% RSLogix 500 project Pump Control HOA and Alarms.RSS, saved by version 8.30.00.16 %
PROJECT "SIM_PLC"    % processor: Bul.1763 MicroLogix 1100 Series B %

PROGRAM FILES
  LAD 2 "MAIN"  4 rungs
  LAD 3 "IO"  11 rungs
  LAD 4 "CTRL LOGIC"  8 rungs
  LAD 5 "ALARMS"  7 rungs

DATA FILES
  O0 OUTPUT  5 elements
  I1 INPUT  7 elements
  S2 STATUS  66 elements
  B3 BINARY  2 elements
  T4 TIMER  4 elements
  C5 COUNTER  1 elements
  R6 CONTROL  1 elements
  N7 INTEGER  4 elements
  F8 FLOAT  1 elements

LADDER 2 "MAIN"
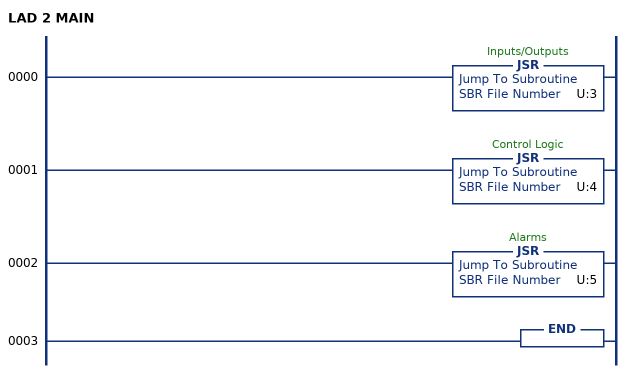
% Rung: 0 %
SOR JSR U:3 EOR
%   U:3  "Inputs/Outputs" %
% Rung: 1 %
SOR JSR U:4 EOR
%   U:4  "Control Logic" %
% Rung: 2 %
SOR JSR U:5 EOR
%   U:5  "Alarms" %
% Rung: 3 %
SOR END EOR

LADDER 3 "IO"
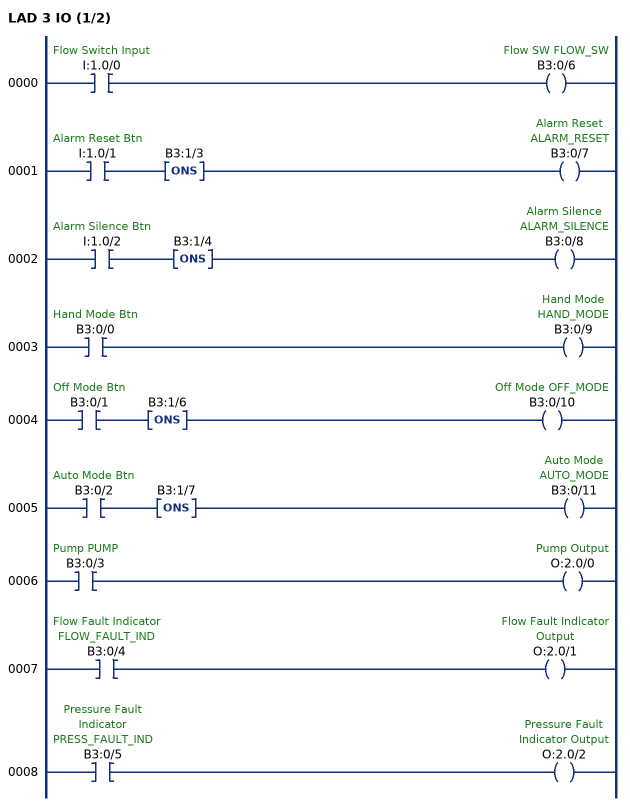
% Rung: 0 %
SOR XIC I:1.0/0 OTE B3:0/6 EOR
%   I:1.0/0  "Flow Switch Input" %
%   B3:0/6  FLOW_SW  "Flow SW" %
% Rung: 1 %
SOR XIC I:1.0/1 ONS B3:1/3 OTE B3:0/7 EOR
%   I:1.0/1  "Alarm Reset Btn" %
%   B3:0/7  ALARM_RESET  "Alarm Reset" %
% Rung: 2 %
SOR XIC I:1.0/2 ONS B3:1/4 OTE B3:0/8 EOR
%   I:1.0/2  "Alarm Silence Btn" %
%   B3:0/8  ALARM_SILENCE  "Alarm Silence" %
% Rung: 3 %
SOR XIC B3:0/0 OTE B3:0/9 EOR
%   B3:0/0  "Hand Mode Btn" %
%   B3:0/9  HAND_MODE  "Hand Mode" %
% Rung: 4 %
SOR XIC B3:0/1 ONS B3:1/6 OTE B3:0/10 EOR
%   B3:0/1  "Off Mode Btn" %
%   B3:0/10  OFF_MODE  "Off Mode" %
% Rung: 5 %
SOR XIC B3:0/2 ONS B3:1/7 OTE B3:0/11 EOR
%   B3:0/2  "Auto Mode Btn" %
%   B3:0/11  AUTO_MODE  "Auto Mode" %
% Rung: 6 %
SOR XIC B3:0/3 OTE O:2.0/0 EOR
%   B3:0/3  PUMP  "Pump" %
%   O:2.0/0  "Pump Output" %
% Rung: 7 %
SOR XIC B3:0/4 OTE O:2.0/1 EOR
%   B3:0/4  FLOW_FAULT_IND  "Flow Fault Indicator" %
%   O:2.0/1  "Flow Fault Indicator Output" %
% Rung: 8 %
SOR XIC B3:0/5 OTE O:2.0/2 EOR
%   B3:0/5  PRESS_FAULT_IND  "Pressure Fault Indicator" %
%   O:2.0/2  "Pressure Fault Indicator Output" %

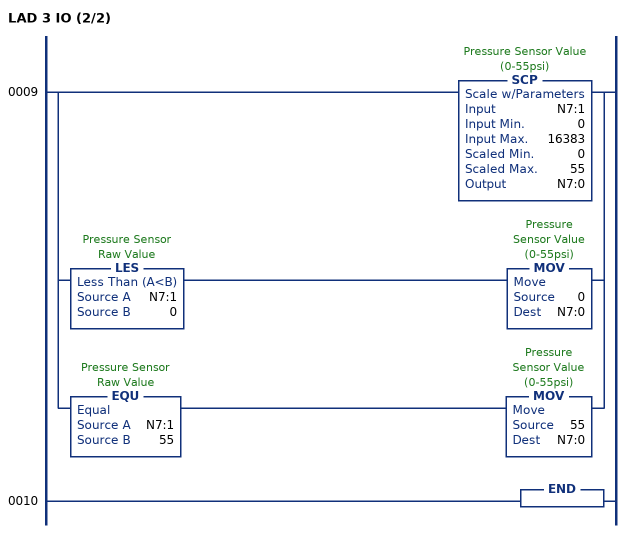
% Rung: 9 %
SOR BST SCP N7:1 0 16383 0 55 N7:0 NXB LES N7:1 0 MOV 0 N7:0 NXB EQU N7:1 55 MOV 55 N7:0 BND EOR
%   N7:1  "Pressure Sensor Raw Value" %
%   N7:0  "Pressure Sensor Value (0-55psi)" %
% Rung: 10 %
SOR END EOR

LADDER 4 "CTRL LOGIC"
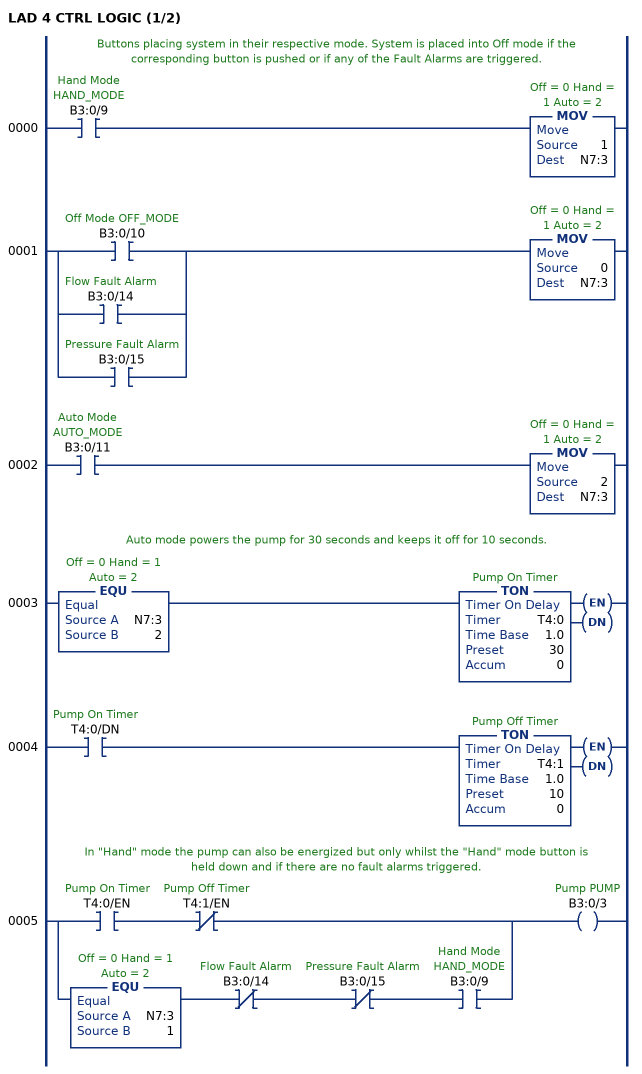
% Rung: 0 %
% Buttons placing system in their respective mode. System is placed into Off mode if the corresponding button is pushed or if any of the Fault Alarms are triggered. %
SOR XIC B3:0/9 MOV 1 N7:3 EOR
%   B3:0/9  HAND_MODE  "Hand Mode" %
%   N7:3  "Off = 0 Hand = 1 Auto = 2" %
% Rung: 1 %
SOR BST XIC B3:0/10 NXB XIC B3:0/14 NXB XIC B3:0/15 BND MOV 0 N7:3 EOR
%   B3:0/10  OFF_MODE  "Off Mode" %
%   B3:0/14  "Flow Fault Alarm" %
%   B3:0/15  "Pressure Fault Alarm" %
%   N7:3  "Off = 0 Hand = 1 Auto = 2" %
% Rung: 2 %
SOR XIC B3:0/11 MOV 2 N7:3 EOR
%   B3:0/11  AUTO_MODE  "Auto Mode" %
%   N7:3  "Off = 0 Hand = 1 Auto = 2" %
% Rung: 3 %
% Auto mode powers the pump for 30 seconds and keeps it off for 10 seconds. %
SOR EQU N7:3 2 TON T4:0 1.0 30 0 EOR
%   N7:3  "Off = 0 Hand = 1 Auto = 2" %
%   T4:0  "Pump On Timer" %
% Rung: 4 %
SOR XIC T4:0/DN TON T4:1 1.0 10 0 EOR
%   T4:0  "Pump On Timer" %
%   T4:1  "Pump Off Timer" %
% Rung: 5 %
% In "Hand" mode the pump can also be energized but only whilst the "Hand" mode button is held down and if there are no fault alarms triggered. %
SOR BST XIC T4:0/EN XIO T4:1/EN NXB EQU N7:3 1 XIO B3:0/14 XIO B3:0/15 XIC B3:0/9 BND OTE B3:0/3 EOR
%   T4:0  "Pump On Timer" %
%   T4:1  "Pump Off Timer" %
%   N7:3  "Off = 0 Hand = 1 Auto = 2" %
%   B3:0/14  "Flow Fault Alarm" %
%   B3:0/15  "Pressure Fault Alarm" %
%   B3:0/9  HAND_MODE  "Hand Mode" %
%   B3:0/3  PUMP  "Pump" %

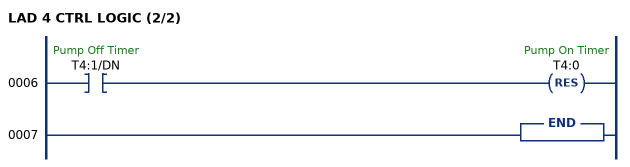
% Rung: 6 %
SOR XIC T4:1/DN RES T4:0 EOR
%   T4:1  "Pump Off Timer" %
%   T4:0  "Pump On Timer" %
% Rung: 7 %
SOR END EOR

LADDER 5 "ALARMS"
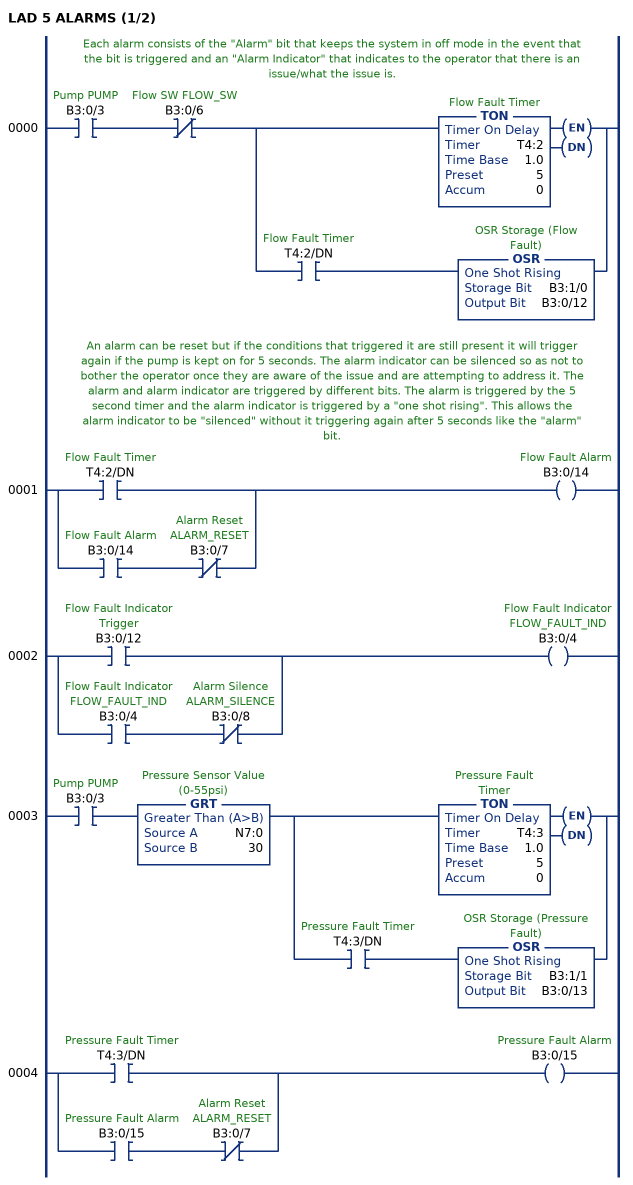
% Rung: 0 %
% Each alarm consists of the "Alarm" bit that keeps the system in off mode in the event that the bit is triggered and an "Alarm Indicator" that indicates to the operator that there is an issue/what the issue is. %
SOR XIC B3:0/3 XIO B3:0/6 BST TON T4:2 1.0 5 0 NXB XIC T4:2/DN OSR B3:1/0 B3:0/12 BND EOR
%   B3:0/3  PUMP  "Pump" %
%   B3:0/6  FLOW_SW  "Flow SW" %
%   T4:2  "Flow Fault Timer" %
%   B3:1/0  "OSR Storage (Flow Fault)" %
%   B3:0/12  "Flow Fault Indicator Trigger" %
% Rung: 1 %
% An alarm can be reset but if the conditions that triggered it are still present it will trigger again if the pump is kept on for 5 seconds. The alarm indicator can be silenced so as not to bother the operator once they are aware of the issue and are attempting to address it. The alarm and alarm indicator are triggered by different bits. The alarm is triggered by the 5 second timer and the alarm indicator is triggered by a "one shot rising". This allows the alarm indicator to be "silenced" without it triggering again after 5 seconds like the "alarm" bit. %
SOR BST XIC T4:2/DN NXB XIC B3:0/14 XIO B3:0/7 BND OTE B3:0/14 EOR
%   T4:2  "Flow Fault Timer" %
%   B3:0/14  "Flow Fault Alarm" %
%   B3:0/7  ALARM_RESET  "Alarm Reset" %
% Rung: 2 %
SOR BST XIC B3:0/12 NXB XIC B3:0/4 XIO B3:0/8 BND OTE B3:0/4 EOR
%   B3:0/12  "Flow Fault Indicator Trigger" %
%   B3:0/4  FLOW_FAULT_IND  "Flow Fault Indicator" %
%   B3:0/8  ALARM_SILENCE  "Alarm Silence" %
% Rung: 3 %
SOR XIC B3:0/3 GRT N7:0 30 BST TON T4:3 1.0 5 0 NXB XIC T4:3/DN OSR B3:1/1 B3:0/13 BND EOR
%   B3:0/3  PUMP  "Pump" %
%   N7:0  "Pressure Sensor Value (0-55psi)" %
%   T4:3  "Pressure Fault Timer" %
%   B3:1/1  "OSR Storage (Pressure Fault)" %
%   B3:0/13  "Pressure Fault Indicator Trigger" %
% Rung: 4 %
SOR BST XIC T4:3/DN NXB XIC B3:0/15 XIO B3:0/7 BND OTE B3:0/15 EOR
%   T4:3  "Pressure Fault Timer" %
%   B3:0/15  "Pressure Fault Alarm" %
%   B3:0/7  ALARM_RESET  "Alarm Reset" %

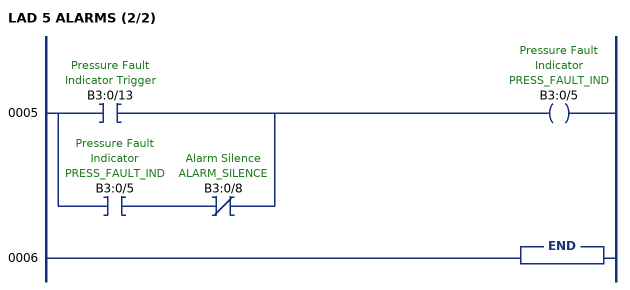
% Rung: 5 %
SOR BST XIC B3:0/13 NXB XIC B3:0/5 XIO B3:0/8 BND OTE B3:0/5 EOR
%   B3:0/13  "Pressure Fault Indicator Trigger" %
%   B3:0/5  PRESS_FAULT_IND  "Pressure Fault Indicator" %
%   B3:0/8  ALARM_SILENCE  "Alarm Silence" %
% Rung: 6 %
SOR END EOR

OTHER DOCUMENTED ADDRESSES
  N7:2  "Hand Mode = 1 Auto or Off = 0"

DATA TABLE (non-zero values as saved)
DATA T4
% .PRE .ACC %
% T4:0 % 30 0
% T4:1 % 10 0
% T4:2 % 5 0
% T4:3 % 5 0
